{attribute addProperty BoxType "AMP8000-0000-0103-0103"}
{attribute addProperty Id "Power_supply_controlwordAT %Q*UINT162"}
{attribute addProperty CRC "4042044998"}
{attribute addProperty SizeInBites "16"}
{attribute addProperty SizeInBytes "2"}
TYPE DeviceMain_Outputs_F0ECB646 :
STRUCT
	{attribute addProperty Name "Power_supply_controlword"}
	Power_supply_controlword AT %Q* : UINT;
END_STRUCT
END_TYPE

(* stored: Version 1.2.0.0, ProductVersion 3.1.4024.9
   DUT DeviceMain_Outputs_F0ECB646: Id {957360ef-4486-455d-aa38-49232fec0218} *)
